(* Logix 5000 project; controller Drives_Line1 1756-L72 rev 20.13; software revision 20.04; part 13 of 21 *)
(* tags used below, declared in another part *)
   Bridle_01 : UDT_Bridle_3M;
   Entry_Accu : UDT_Entry_Accu;
   EntryConfig : UDT_Config_Zone;
   EntryCtrl : UDT_Control_Zone;
   EntrySetpoints : UDT_Setpoints_Zone;
   EntryStat : UDT_Status_Zone;
   In_Commands : UDT_Commands;
   In_Config : UDT_Config;
   In_Setpoints : UDT_Setpoints;
   LineCmd : UDT_Commands_Line;
   LineCtrl : UDT_Control_Line;
   LineStat : UDT_Status_Line;
   TM1 : UDT_TM;
   zConfigFromMaster : BOOL;

PROGRAM P16_Entry_Accu   (* main routine R00_Main *)
VAR
   ABS_01 : FBD_MATH_ADVANCED := (Source := -0.00068994303, Dest := 0.00068994303);
   BAND_01 : FBD_BOOLEAN_AND := (In3 := 1, In4 := 1, In5 := 1, In6 := 1, In7 := 1, In8 := 1);
   BAND_03 : FBD_BOOLEAN_AND := (In3 := 1, In4 := 1, In5 := 1, In6 := 1, In7 := 1, In8 := 1);
   BNOT_01 : FBD_BOOLEAN_NOT := (Out := 1);
   BNOT_02 : FBD_BOOLEAN_NOT := (In := 1);
   BNOT_04 : FBD_BOOLEAN_NOT := (Out := 1);
   BNOT_06 : FBD_BOOLEAN_NOT := (Out := 1);
   BOR_01 : FBD_BOOLEAN_OR;
   DIV_01 : FBD_MATH := (SourceA := -0.00068994303, SourceB := 4.0, Dest := -0.00017248576);
   DIV_02 : FBD_MATH;
   DIV_03 : FBD_MATH := (SourceA := 2.0441563, SourceB := 100.0, Dest := 0.020441564);
   DIV_04 : FBD_MATH := (SourceA := 0.5, SourceB := 4.0, Dest := 0.125);
   Entry_Accu_FBCounts_mm : DINT := 742;
   Entry_Accu_rev_mm : REAL := 0.1811;
   Exit_Accu_Rev_mm : REAL := 5.030181;
   IO_State_Exit_Accu : INT := 4;
   IO_State_Tmp_Exit_Accu : INT := 16384;
   MUL_01 : FBD_MATH := (SourceA := -2.9323564e-07, SourceB := 10865.999, Dest := -0.0031862983);
   MUL_02 : FBD_MATH := (SourceA := 2.0, SourceB := 2.0, Dest := 4.0);
   MUL_03 : FBD_MATH := (SourceA := 11670.0, SourceB := 742.0, Dest := 8659140.0);
   MUL_04 : FBD_MATH := (SourceB := 742.0);
   MUL_05 : FBD_MATH := (SourceA := 0.00034438504, SourceB := 0.5, Dest := 0.00017219252);
   MUL_06 : FBD_MATH := (SourceA := 1000.0, SourceB := 0.1811, Dest := 181.09999);
   MUL_07 : FBD_MATH := (SourceA := 181.09999, SourceB := 60.0, Dest := 10865.999);
   NEG_01 : FBD_MATH_ADVANCED := (Source := 50.0, Dest := -50.0);
   NEG_04 : FBD_MATH_ADVANCED := (Source := 0.02, Dest := -0.02);
   NEG_06 : FBD_MATH_ADVANCED := (Source := 0.020441564, Dest := -0.020441564);
   ons : BOOL[32];
   PI_01 : PROP_INT := (In := 23.319267, Initialize := 1, Kp := 25.0, Wld := 0.075, HighLimit := 100.0, ShapeKpPlus := 1.0, ShapeKpMinus := 1.0, ShapeWldPlus := 1.0, ShapeWldMinus := 1.0, RTSTime := 1, LowAlarm := 1, DeltaT := 0.05);
   PI_02 : PROP_INT := (In := -0.00033332407, Kp := 0.085, Wld := 0.01, HighLimit := 0.020441564, LowLimit := -0.020441564, ShapeKpPlus := 1.0, ShapeKpMinus := 1.0, ShapeWldPlus := 1.0, ShapeWldMinus := 1.0, RTSTime := 1, Out := 0.0003160029, DeltaT := 0.05);
   RLIM_01 : RATE_LIMITER := (In := -0.00017248576, IncRate := 0.5, DecRate := 0.5, RTSTime := 1, Out := -0.00017248576, DeltaT := 0.05);
   SCL_01 : SCALE := (In := 6033752.0, InRawMax := 8659140.0, InEUMax := 100.0, Out := 69.68073);
   SCL_02 : SCALE := (In := 6033752.0, InRawMax := 8659140.0, InEUMax := 11670.0, Out := 8131.741);
   SCL_03 : SCALE := (InRawMax := 100.0, Limiting := 1);
   SCL_04 : SCALE := (In := 5850.0, InRawMax := 30000.0, InEUMax := 1.0, Limiting := 1, Out := 0.19500001);
   SCL_05 : SCALE := (In := 5860.0, InRawMax := 30000.0, InEUMax := 1.0, Out := 0.19533333);
   SCL_08 : SCALE := (In := 0.00068994303, InRawMax := 0.125, InEUMax := 10.0, InEUMin := 2.0, Limiting := 1, Out := 2.0441563);
   SCRV_01 : S_CURVE := (Initialize := 1, AbsAlgRamp := 1, AccelRate := 0.04, DecelRate := 0.04, JerkRate := 0.25, RTSTime := 1, DeltaT := 0.05);
   SEL_01 : SELECT := (In1 := 50.0, In2 := 20.0, Out := 50.0);
   SSUM_01 : SELECTED_SUMMER := (In1 := 0.02, Gain1 := 1.0, In2 := -0.02, Gain2 := 1.0, Gain3 := 1.0, Select3 := 1, Gain4 := 1.0, Gain5 := 1.0, Gain6 := 1.0, Gain7 := 1.0, Gain8 := 1.0);
   SSUM_03 : SELECTED_SUMMER := (In1 := -0.00017248576, Gain1 := 1.0, Select1 := 1, Gain2 := 1.0, Gain3 := 1.0, Gain4 := 1.0, Gain5 := 1.0, Gain6 := 1.0, Gain7 := 1.0, Gain8 := 1.0, Out := -0.00017248576);
   SSUM_05 : SELECTED_SUMMER := (In1 := 0.00017219252, Gain1 := 1.0, Select1 := 1, In2 := -0.00017248576, Gain2 := 1.0, Select2 := 1, Gain3 := 1.0, Gain4 := 1.0, Gain5 := 1.0, Gain6 := 1.0, Gain7 := 1.0, Gain8 := 1.0, Out := -2.9323564e-07);
   SUB_01 : FBD_MATH := (SourceA := 93.0, SourceB := 69.68073, Dest := 23.319267);
   SUB_02 : FBD_MATH := (SourceA := 0.19500001, SourceB := 0.19533333, Dest := -0.00033332407);
   SUB_03 : FBD_MATH := (SourceB := 0.00068994303, Dest := -0.00068994303);
   SUB_04 : FBD_MATH := (SourceB := 0.00068994303, Dest := -0.00068994303);
   TofReset : TIMER := (PRE := 1000, ACC := 1000);
   TofTensionOnSp : TIMER := (PRE := 2500, ACC := 2500);
   TonNoResponse : TIMER := (PRE := 2500);
   TonRefOn : TIMER := (PRE := 750);
   TonTensionOnSp : TIMER := (PRE := 500, ACC := 549, EN := 1, DN := 1);
   zEntry_Accu_EncCounts : DINT := 4096;
   zEntry_Accu_Kp_Treg : REAL := 0.085;
   zEntry_Accu_MaxAccDec : REAL := 0.5;
   zEntry_Accu_Pos_PreLim : REAL := 100.0;
   zEntry_Accu_SpdRegMax : REAL := 50.0;
   zEntry_Accu_SpdRegMin : REAL := 20.0;
   zEntry_Accu_SpdTrim_HL : REAL := 10.0;
   zEntry_Accu_SpdTrim_LL : REAL := 2.0;
   zEntry_Accu_WLD_Treg : REAL := 0.01;
   zExit_Accu_Kp_Preg : REAL := 25.0;
   zExit_Accu_WLD_Preg : REAL := 0.075;
   zNoMaster : BOOL := 1;
   zTM1_Tens_Offset : REAL := 500.0;
END_VAR

ROUTINE R00_Main   (* ladder *)
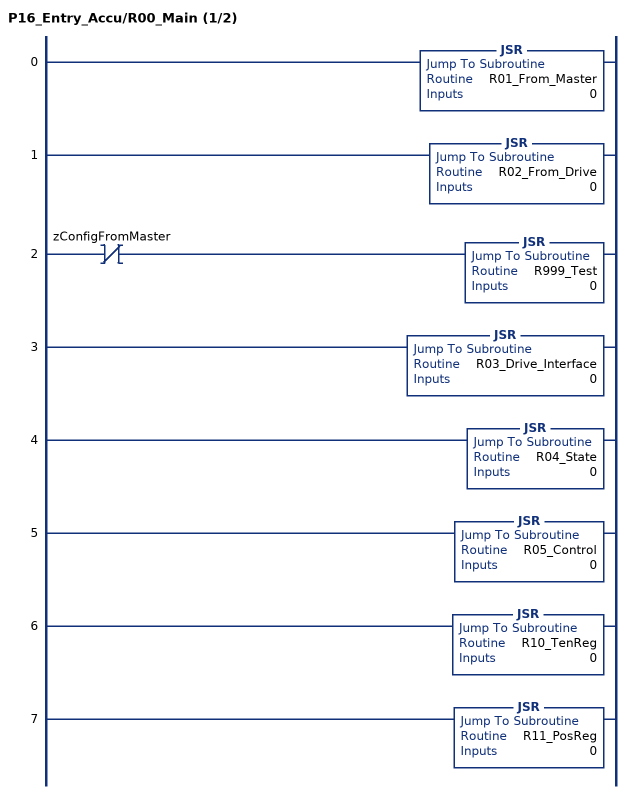
   0: JSR(R01_From_Master,0);
   1: JSR(R02_From_Drive,0);
   2: XIO(zConfigFromMaster)JSR(R999_Test,0);
   3: JSR(R03_Drive_Interface,0);
   4: JSR(R04_State,0);
   5: JSR(R05_Control,0);
   6: JSR(R10_TenReg,0);
   7: JSR(R11_PosReg,0);
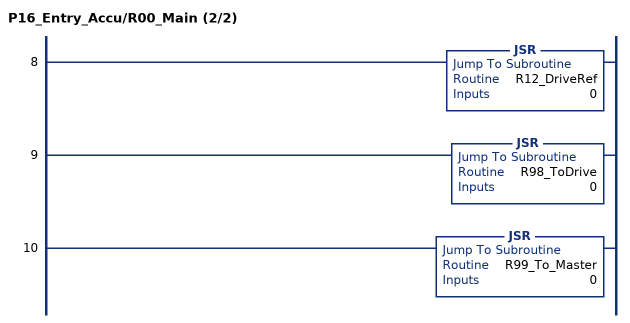
   8: JSR(R12_DriveRef,0);
   9: JSR(R98_ToDrive,0);
   10: JSR(R99_To_Master,0);
END_ROUTINE

ROUTINE R01_From_Master   (* ladder *)
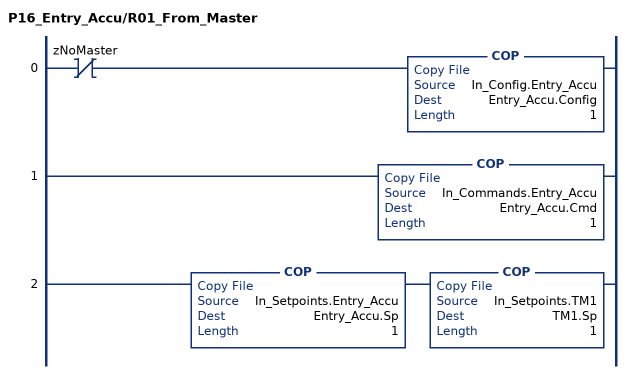
   0: XIO(zNoMaster)COP(In_Config.Entry_Accu,Entry_Accu.Config,1);
   1: COP(In_Commands.Entry_Accu,Entry_Accu.Cmd,1);
   2: COP(In_Setpoints.Entry_Accu,Entry_Accu.Sp,1)COP(In_Setpoints.TM1,TM1.Sp,1);
END_ROUTINE

ROUTINE R02_From_Drive   (* ladder *)
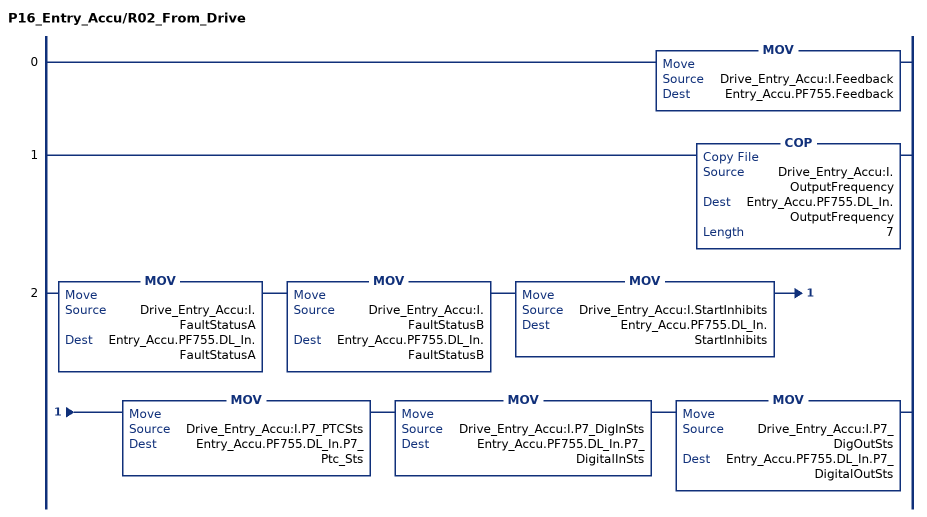
   0: MOV(Drive_Entry_Accu:I.Feedback,Entry_Accu.PF755.Feedback);
   1: COP(Drive_Entry_Accu:I.OutputFrequency,Entry_Accu.PF755.DL_In.OutputFrequency,7);
   2: MOV(Drive_Entry_Accu:I.FaultStatusA,Entry_Accu.PF755.DL_In.FaultStatusA)MOV(Drive_Entry_Accu:I.FaultStatusB,Entry_Accu.PF755.DL_In.FaultStatusB)MOV(Drive_Entry_Accu:I.StartInhibits,Entry_Accu.PF755.DL_In.StartInhibits)MOV(Drive_Entry_Accu:I.P7_PTCSts,Entry_Accu.PF755.DL_In.P7_Ptc_Sts)MOV(Drive_Entry_Accu:I.P7_DigInSts,Entry_Accu.PF755.DL_In.P7_DigitalInSts)MOV(Drive_Entry_Accu:I.P7_DigOutSts,Entry_Accu.PF755.DL_In.P7_DigitalOutSts);
END_ROUTINE

ROUTINE R03_Drive_Interface   (* ladder *)
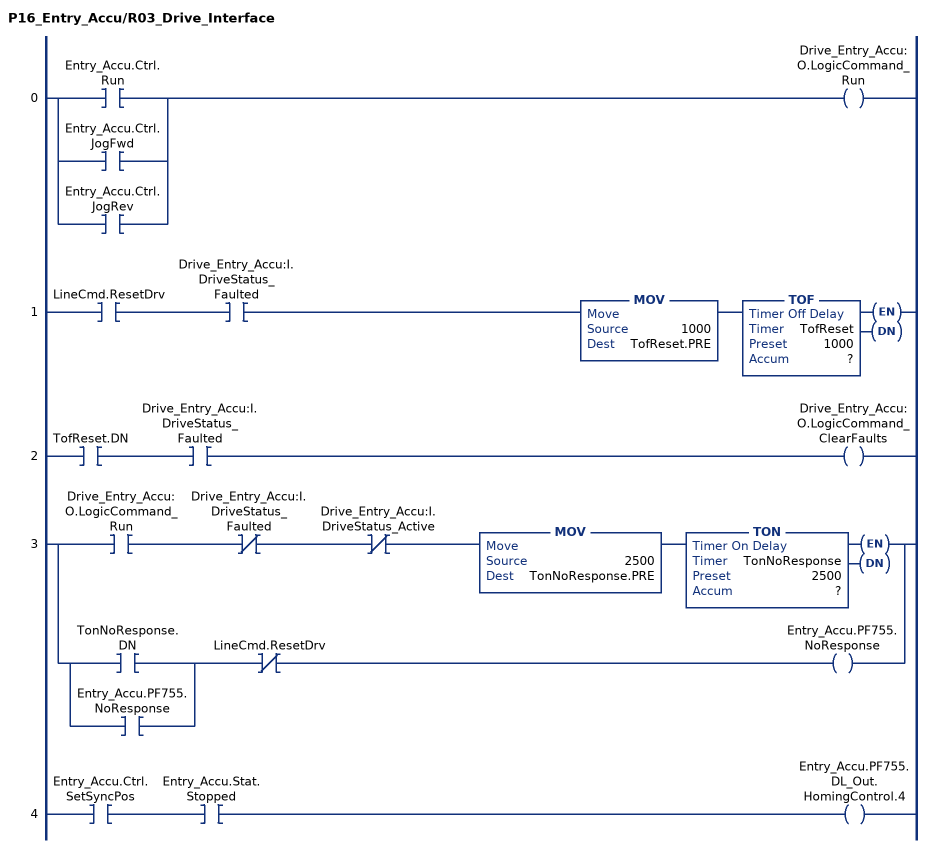
   0: [XIC(Entry_Accu.Ctrl.Run) ,XIC(Entry_Accu.Ctrl.JogFwd) ,XIC(Entry_Accu.Ctrl.JogRev) ]OTE(Drive_Entry_Accu:O.LogicCommand_Run);
   1: XIC(LineCmd.ResetDrv)XIC(Drive_Entry_Accu:I.DriveStatus_Faulted)MOV(1000,TofReset.PRE)TOF(TofReset,?,?);
   2: XIC(TofReset.DN)XIC(Drive_Entry_Accu:I.DriveStatus_Faulted)OTE(Drive_Entry_Accu:O.LogicCommand_ClearFaults);
   3: [XIC(Drive_Entry_Accu:O.LogicCommand_Run) XIO(Drive_Entry_Accu:I.DriveStatus_Faulted) XIO(Drive_Entry_Accu:I.DriveStatus_Active) MOV(2500,TonNoResponse.PRE) TON(TonNoResponse,?,?) ,[XIC(TonNoResponse.DN) ,XIC(Entry_Accu.PF755.NoResponse) ] XIO(LineCmd.ResetDrv) OTE(Entry_Accu.PF755.NoResponse) ];
   4: XIC(Entry_Accu.Ctrl.SetSyncPos)XIC(Entry_Accu.Stat.Stopped)OTE(Entry_Accu.PF755.DL_Out.HomingControl.4);
END_ROUTINE

ROUTINE R04_State   (* ladder *)
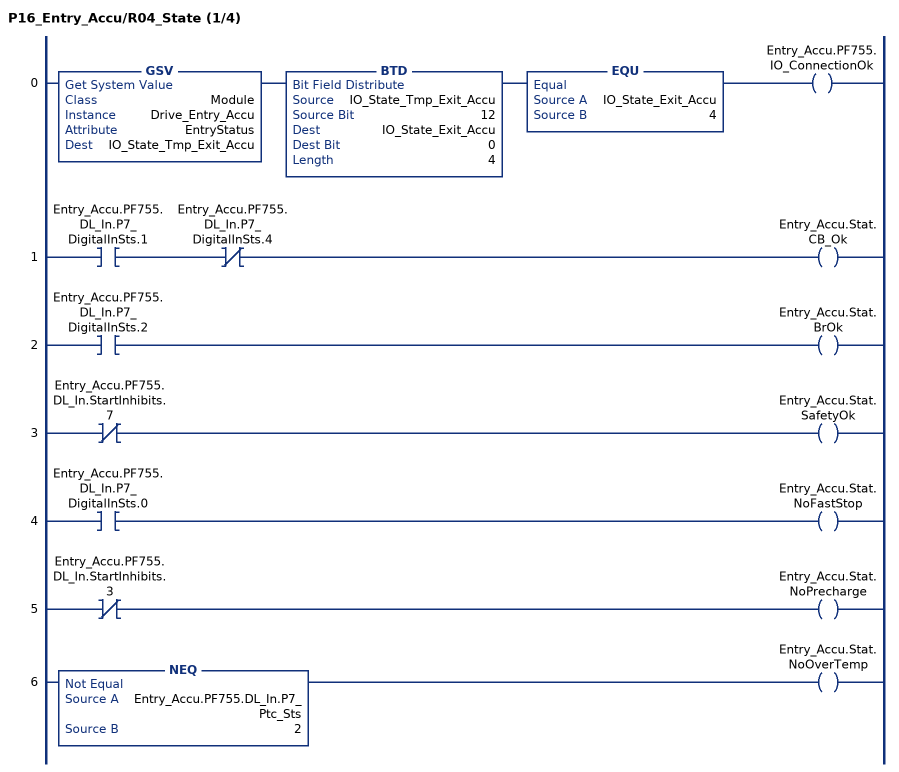
   0: GSV(Module,Drive_Entry_Accu,EntryStatus,IO_State_Tmp_Exit_Accu)BTD(IO_State_Tmp_Exit_Accu,12,IO_State_Exit_Accu,0,4)EQU(IO_State_Exit_Accu,4)OTE(Entry_Accu.PF755.IO_ConnectionOk);
   1: XIC(Entry_Accu.PF755.DL_In.P7_DigitalInSts.1)XIO(Entry_Accu.PF755.DL_In.P7_DigitalInSts.4)OTE(Entry_Accu.Stat.CB_Ok);
   2: XIC(Entry_Accu.PF755.DL_In.P7_DigitalInSts.2)OTE(Entry_Accu.Stat.BrOk);
   3: XIO(Entry_Accu.PF755.DL_In.StartInhibits.7)OTE(Entry_Accu.Stat.SafetyOk);
   4: XIC(Entry_Accu.PF755.DL_In.P7_DigitalInSts.0)OTE(Entry_Accu.Stat.NoFastStop);
   5: XIO(Entry_Accu.PF755.DL_In.StartInhibits.3)OTE(Entry_Accu.Stat.NoPrecharge);
   6: NEQ(Entry_Accu.PF755.DL_In.P7_Ptc_Sts,2)OTE(Entry_Accu.Stat.NoOverTemp);
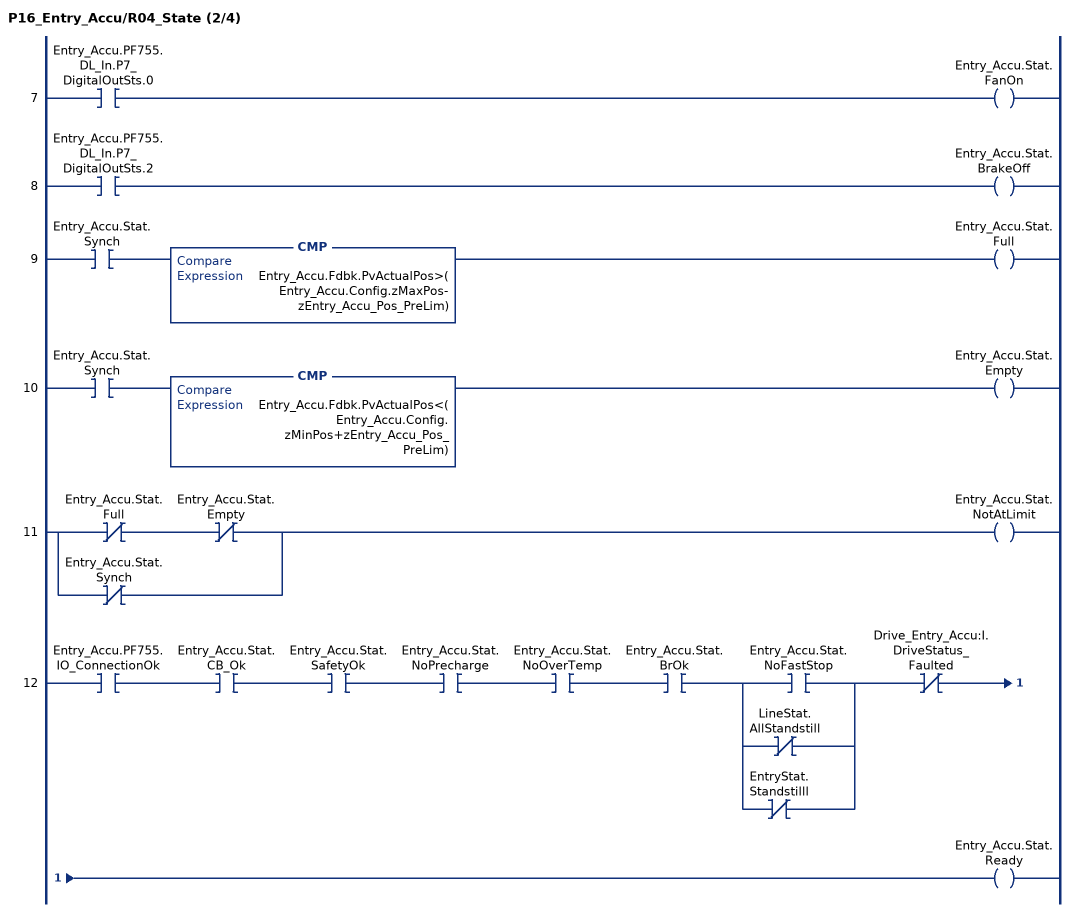
   7: XIC(Entry_Accu.PF755.DL_In.P7_DigitalOutSts.0)OTE(Entry_Accu.Stat.FanOn);
   8: XIC(Entry_Accu.PF755.DL_In.P7_DigitalOutSts.2)OTE(Entry_Accu.Stat.BrakeOff);
   9: XIC(Entry_Accu.Stat.Synch)CMP(Entry_Accu.Fdbk.PvActualPos>(Entry_Accu.Config.zMaxPos-zEntry_Accu_Pos_PreLim))OTE(Entry_Accu.Stat.Full);
   10: XIC(Entry_Accu.Stat.Synch)CMP(Entry_Accu.Fdbk.PvActualPos<(Entry_Accu.Config.zMinPos+zEntry_Accu_Pos_PreLim))OTE(Entry_Accu.Stat.Empty);
   11: [XIO(Entry_Accu.Stat.Full) XIO(Entry_Accu.Stat.Empty) ,XIO(Entry_Accu.Stat.Synch) ]OTE(Entry_Accu.Stat.NotAtLimit);
   12: XIC(Entry_Accu.PF755.IO_ConnectionOk)XIC(Entry_Accu.Stat.CB_Ok)XIC(Entry_Accu.Stat.SafetyOk)XIC(Entry_Accu.Stat.NoPrecharge)XIC(Entry_Accu.Stat.NoOverTemp)XIC(Entry_Accu.Stat.BrOk)[XIC(Entry_Accu.Stat.NoFastStop) ,XIO(LineStat.AllStandstill) ,XIO(EntryStat.Standstilll) ]XIO(Drive_Entry_Accu:I.DriveStatus_Faulted)OTE(Entry_Accu.Stat.Ready);
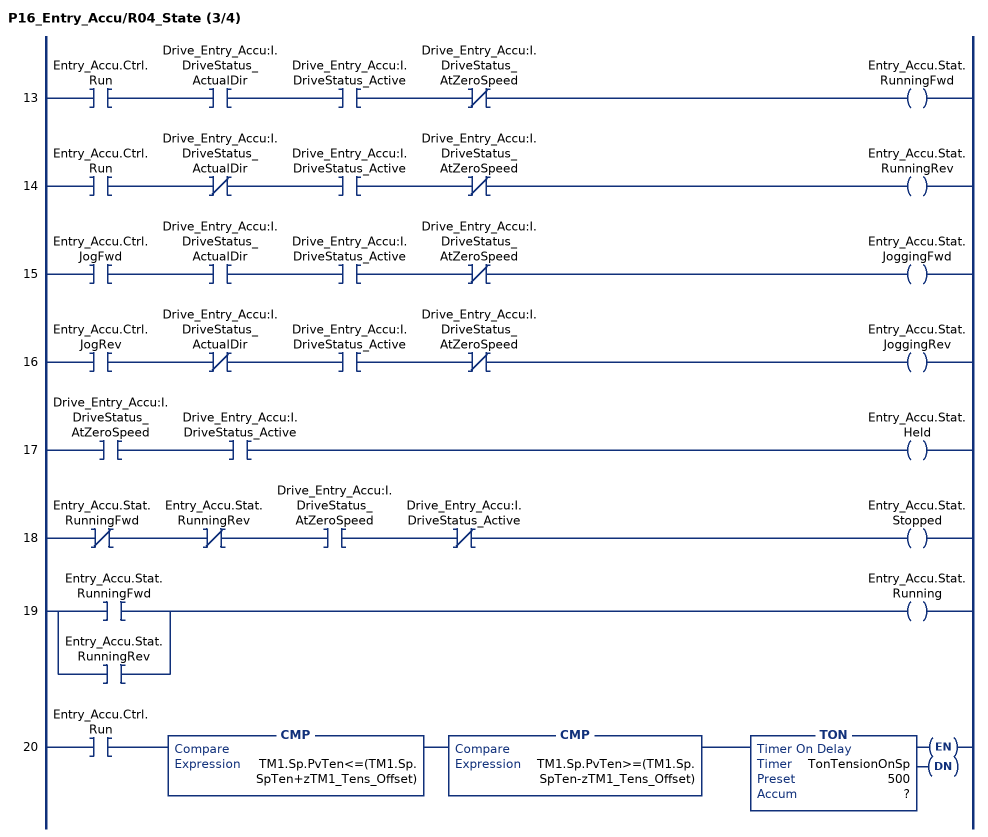
   13: XIC(Entry_Accu.Ctrl.Run)XIC(Drive_Entry_Accu:I.DriveStatus_ActualDir)XIC(Drive_Entry_Accu:I.DriveStatus_Active)XIO(Drive_Entry_Accu:I.DriveStatus_AtZeroSpeed)OTE(Entry_Accu.Stat.RunningFwd);
   14: XIC(Entry_Accu.Ctrl.Run)XIO(Drive_Entry_Accu:I.DriveStatus_ActualDir)XIC(Drive_Entry_Accu:I.DriveStatus_Active)XIO(Drive_Entry_Accu:I.DriveStatus_AtZeroSpeed)OTE(Entry_Accu.Stat.RunningRev);
   15: XIC(Entry_Accu.Ctrl.JogFwd)XIC(Drive_Entry_Accu:I.DriveStatus_ActualDir)XIC(Drive_Entry_Accu:I.DriveStatus_Active)XIO(Drive_Entry_Accu:I.DriveStatus_AtZeroSpeed)OTE(Entry_Accu.Stat.JoggingFwd);
   16: XIC(Entry_Accu.Ctrl.JogRev)XIO(Drive_Entry_Accu:I.DriveStatus_ActualDir)XIC(Drive_Entry_Accu:I.DriveStatus_Active)XIO(Drive_Entry_Accu:I.DriveStatus_AtZeroSpeed)OTE(Entry_Accu.Stat.JoggingRev);
   17: XIC(Drive_Entry_Accu:I.DriveStatus_AtZeroSpeed)XIC(Drive_Entry_Accu:I.DriveStatus_Active)OTE(Entry_Accu.Stat.Held);
   18: XIO(Entry_Accu.Stat.RunningFwd)XIO(Entry_Accu.Stat.RunningRev)XIC(Drive_Entry_Accu:I.DriveStatus_AtZeroSpeed)XIO(Drive_Entry_Accu:I.DriveStatus_Active)OTE(Entry_Accu.Stat.Stopped);
   19: [XIC(Entry_Accu.Stat.RunningFwd) ,XIC(Entry_Accu.Stat.RunningRev) ]OTE(Entry_Accu.Stat.Running);
   20: XIC(Entry_Accu.Ctrl.Run)CMP(TM1.Sp.PvTen<=(TM1.Sp.SpTen+zTM1_Tens_Offset))CMP(TM1.Sp.PvTen>=(TM1.Sp.SpTen-zTM1_Tens_Offset))TON(TonTensionOnSp,?,?);
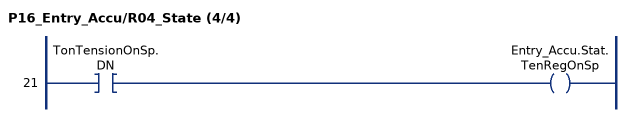
   21: XIC(TonTensionOnSp.DN)OTE(Entry_Accu.Stat.TenRegOnSp);
END_ROUTINE

ROUTINE R05_Control   (* ladder *)
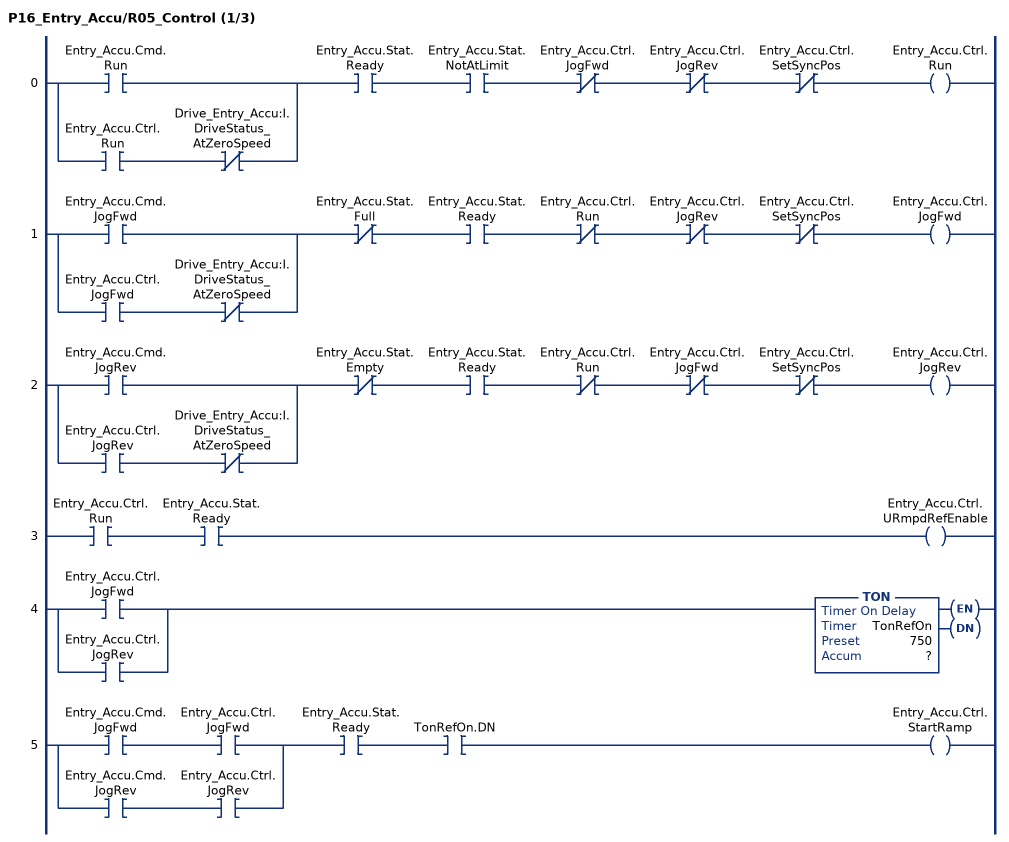
   0: [XIC(Entry_Accu.Cmd.Run) ,XIC(Entry_Accu.Ctrl.Run) XIO(Drive_Entry_Accu:I.DriveStatus_AtZeroSpeed) ]XIC(Entry_Accu.Stat.Ready)XIC(Entry_Accu.Stat.NotAtLimit)XIO(Entry_Accu.Ctrl.JogFwd)XIO(Entry_Accu.Ctrl.JogRev)XIO(Entry_Accu.Ctrl.SetSyncPos)OTE(Entry_Accu.Ctrl.Run);
   1: [XIC(Entry_Accu.Cmd.JogFwd) ,XIC(Entry_Accu.Ctrl.JogFwd) XIO(Drive_Entry_Accu:I.DriveStatus_AtZeroSpeed) ]XIO(Entry_Accu.Stat.Full)XIC(Entry_Accu.Stat.Ready)XIO(Entry_Accu.Ctrl.Run)XIO(Entry_Accu.Ctrl.JogRev)XIO(Entry_Accu.Ctrl.SetSyncPos)OTE(Entry_Accu.Ctrl.JogFwd);
   2: [XIC(Entry_Accu.Cmd.JogRev) ,XIC(Entry_Accu.Ctrl.JogRev) XIO(Drive_Entry_Accu:I.DriveStatus_AtZeroSpeed) ]XIO(Entry_Accu.Stat.Empty)XIC(Entry_Accu.Stat.Ready)XIO(Entry_Accu.Ctrl.Run)XIO(Entry_Accu.Ctrl.JogFwd)XIO(Entry_Accu.Ctrl.SetSyncPos)OTE(Entry_Accu.Ctrl.JogRev);
   3: XIC(Entry_Accu.Ctrl.Run)XIC(Entry_Accu.Stat.Ready)OTE(Entry_Accu.Ctrl.URmpdRefEnable);
   4: [XIC(Entry_Accu.Ctrl.JogFwd) ,XIC(Entry_Accu.Ctrl.JogRev) ]TON(TonRefOn,?,?);
   5: [XIC(Entry_Accu.Cmd.JogFwd) XIC(Entry_Accu.Ctrl.JogFwd) ,XIC(Entry_Accu.Cmd.JogRev) XIC(Entry_Accu.Ctrl.JogRev) ]XIC(Entry_Accu.Stat.Ready)XIC(TonRefOn.DN)OTE(Entry_Accu.Ctrl.StartRamp);
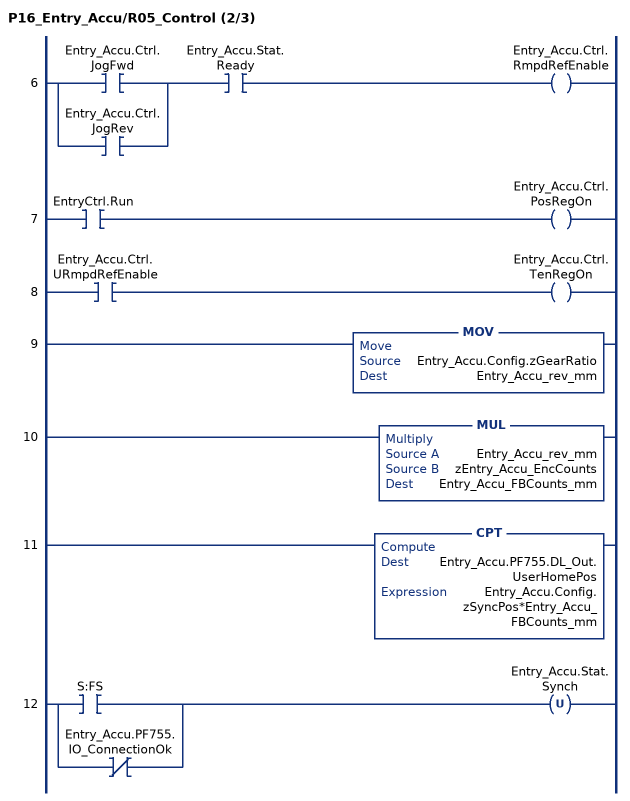
   6: [XIC(Entry_Accu.Ctrl.JogFwd) ,XIC(Entry_Accu.Ctrl.JogRev) ]XIC(Entry_Accu.Stat.Ready)OTE(Entry_Accu.Ctrl.RmpdRefEnable);
   7: XIC(EntryCtrl.Run)OTE(Entry_Accu.Ctrl.PosRegOn);
   8: XIC(Entry_Accu.Ctrl.URmpdRefEnable)OTE(Entry_Accu.Ctrl.TenRegOn);
   9: MOV(Entry_Accu.Config.zGearRatio,Entry_Accu_rev_mm);
   10: MUL(Entry_Accu_rev_mm,zEntry_Accu_EncCounts,Entry_Accu_FBCounts_mm);
   11: CPT(Entry_Accu.PF755.DL_Out.UserHomePos,Entry_Accu.Config.zSyncPos*Entry_Accu_FBCounts_mm);
   12: [XIC(S:FS) ,XIO(Entry_Accu.PF755.IO_ConnectionOk) ]OTU(Entry_Accu.Stat.Synch);
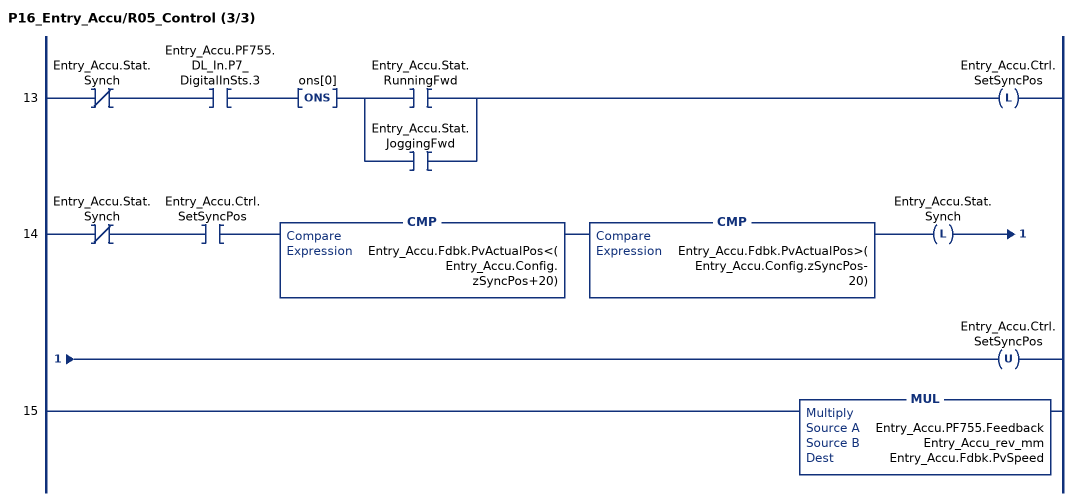
   13: XIO(Entry_Accu.Stat.Synch)XIC(Entry_Accu.PF755.DL_In.P7_DigitalInSts.3)ONS(ons[0])[XIC(Entry_Accu.Stat.RunningFwd) ,XIC(Entry_Accu.Stat.JoggingFwd) ]OTL(Entry_Accu.Ctrl.SetSyncPos);
   14: XIO(Entry_Accu.Stat.Synch)XIC(Entry_Accu.Ctrl.SetSyncPos)CMP(Entry_Accu.Fdbk.PvActualPos<(Entry_Accu.Config.zSyncPos+20))CMP(Entry_Accu.Fdbk.PvActualPos>(Entry_Accu.Config.zSyncPos-20))OTL(Entry_Accu.Stat.Synch)OTU(Entry_Accu.Ctrl.SetSyncPos);
   15: MUL(Entry_Accu.PF755.Feedback,Entry_Accu_rev_mm,Entry_Accu.Fdbk.PvSpeed);
END_ROUTINE

ROUTINE R10_TenReg   (* function block diagram *)
   SHEET 1   // Scale setpoint
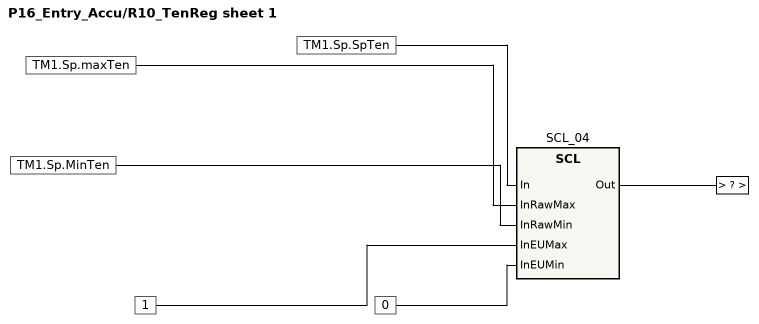
   SCL_04 : SCL(In := TM1.Sp.SpTen, InRawMax := TM1.Sp.maxTen, InRawMin := TM1.Sp.MinTen, InEUMax := 1, InEUMin := 0);
   WIRE(?) := SCL_04.Out;
   SHEET 2   // Scale tension feedback
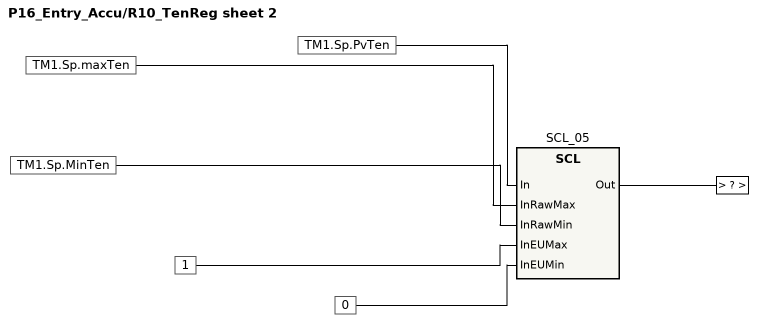
   SCL_05 : SCL(In := TM1.Sp.PvTen, InRawMax := TM1.Sp.maxTen, InRawMin := TM1.Sp.MinTen, InEUMax := 1, InEUMin := 0);
   WIRE(?) := SCL_05.Out;
   SHEET 3   // Trim limits
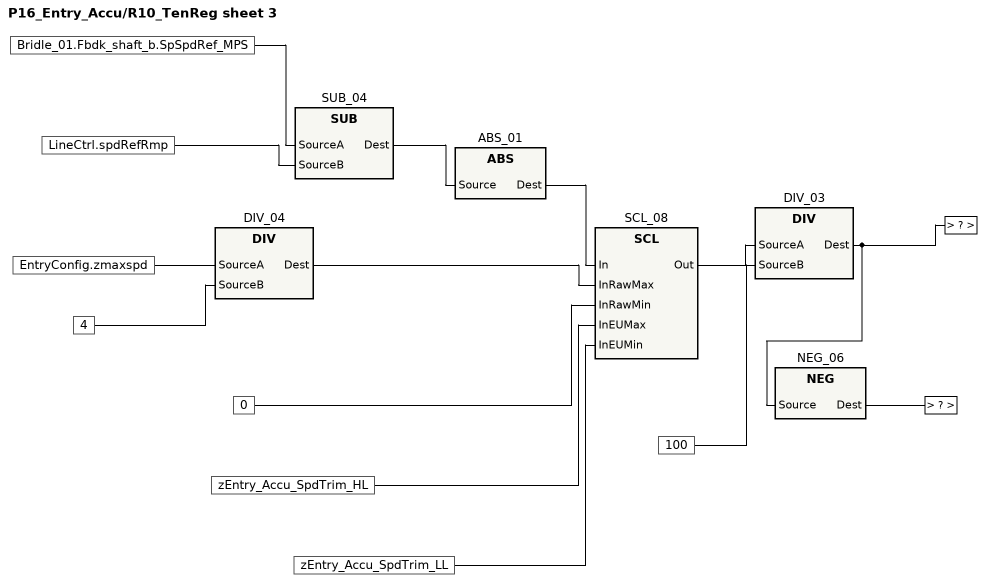
   DIV_04 : DIV(SourceA := EntryConfig.zmaxspd, SourceB := 4);
   SUB_04 : SUB(SourceA := Bridle_01.Fbdk_shaft_b.SpSpdRef_MPS, SourceB := LineCtrl.spdRefRmp);
   ABS_01 : ABS(Source := SUB_04.Dest);
   SCL_08 : SCL(In := ABS_01.Dest, InRawMax := DIV_04.Dest, InRawMin := 0, InEUMax := zEntry_Accu_SpdTrim_HL, InEUMin := zEntry_Accu_SpdTrim_LL);
   DIV_03 : DIV(SourceA := SCL_08.Out, SourceB := 100);
   NEG_06 : NEG(Source := DIV_03.Dest);
   WIRE(?) := NEG_06.Dest;
   WIRE(?) := DIV_03.Dest;
   SHEET 4   // Tension regulator
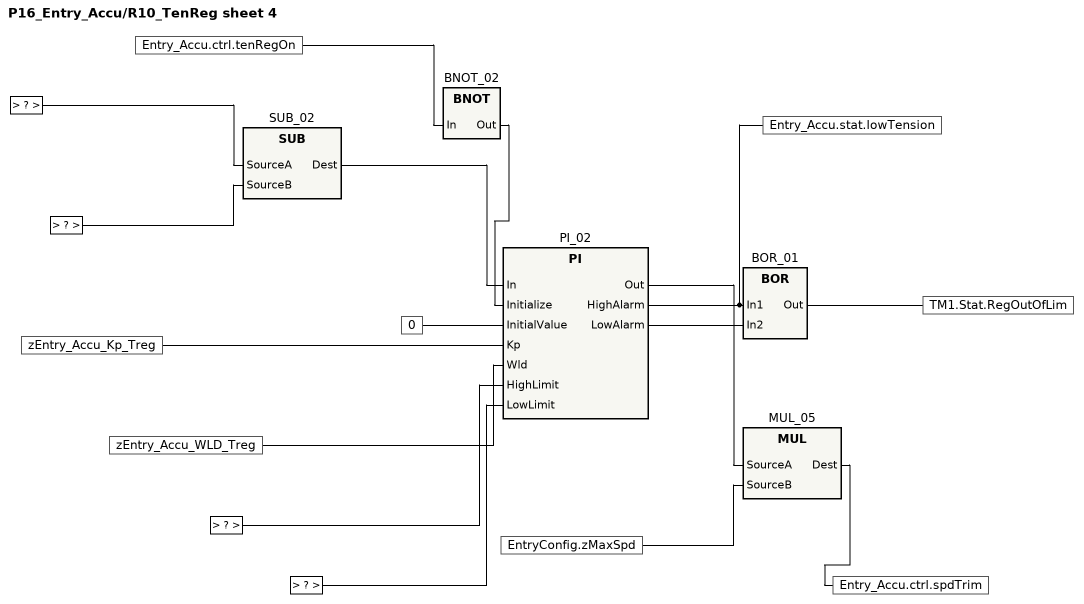
   SUB_02 : SUB(SourceA := WIRE(?), SourceB := WIRE(?));
   BNOT_02 : BNOT(In := Entry_Accu.ctrl.tenRegOn);
   PI_02 : PI(In := SUB_02.Dest, Initialize := BNOT_02.Out, InitialValue := 0, Kp := zEntry_Accu_Kp_Treg, Wld := zEntry_Accu_WLD_Treg, HighLimit := WIRE(?), LowLimit := WIRE(?));
   BOR_01 : BOR(In1 := PI_02.HighAlarm, In2 := PI_02.LowAlarm);
   MUL_05 : MUL(SourceA := PI_02.Out, SourceB := EntryConfig.zMaxSpd);
   Entry_Accu.stat.lowTension := PI_02.HighAlarm;
   Entry_Accu.ctrl.spdTrim := MUL_05.Dest;
   TM1.Stat.RegOutOfLim := BOR_01.Out;
END_ROUTINE

ROUTINE R11_PosReg   (* function block diagram *)
   SHEET 1   // Scale feedback
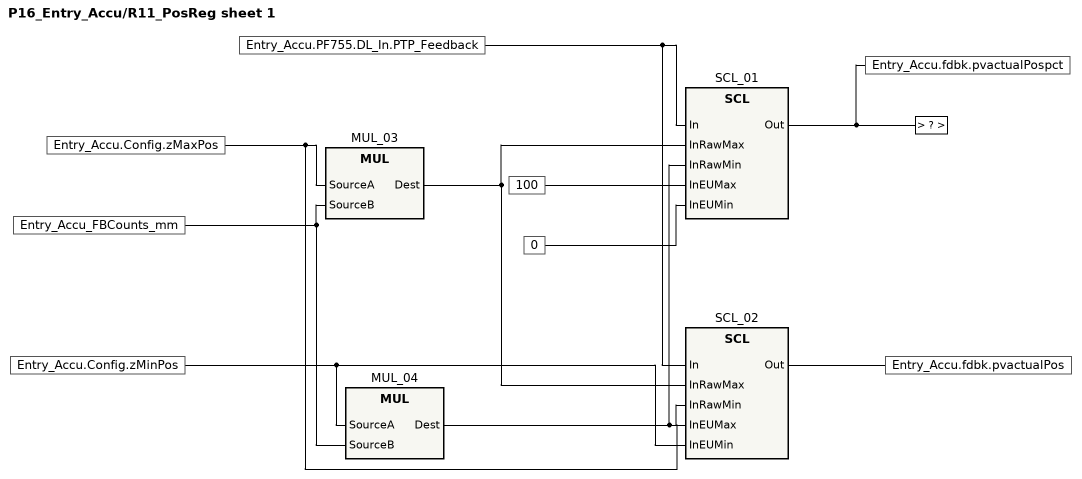
   MUL_03 : MUL(SourceA := Entry_Accu.Config.zMaxPos, SourceB := Entry_Accu_FBCounts_mm);
   MUL_04 : MUL(SourceA := Entry_Accu.Config.zMinPos, SourceB := Entry_Accu_FBCounts_mm);
   SCL_01 : SCL(In := Entry_Accu.PF755.DL_In.PTP_Feedback, InRawMax := MUL_03.Dest, InRawMin := MUL_04.Dest, InEUMax := 100, InEUMin := 0);
   SCL_02 : SCL(In := Entry_Accu.PF755.DL_In.PTP_Feedback, InRawMax := MUL_03.Dest, InRawMin := MUL_04.Dest, InEUMax := Entry_Accu.Config.zMaxPos, InEUMin := Entry_Accu.Config.zMinPos);
   Entry_Accu.fdbk.pvactualPospct := SCL_01.Out;
   Entry_Accu.fdbk.pvactualPos := SCL_02.Out;
   WIRE(?) := SCL_01.Out;
   SHEET 2   // Position regulator
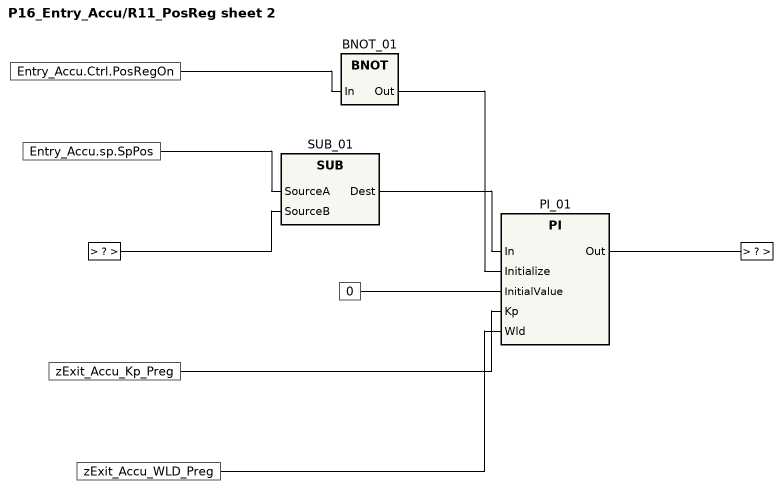
   BNOT_01 : BNOT(In := Entry_Accu.Ctrl.PosRegOn);
   SUB_01 : SUB(SourceA := Entry_Accu.sp.SpPos, SourceB := WIRE(?));
   PI_01 : PI(In := SUB_01.Dest, Initialize := BNOT_01.Out, InitialValue := 0, Kp := zExit_Accu_Kp_Preg, Wld := zExit_Accu_WLD_Preg);
   WIRE(?) := PI_01.Out;
   SHEET 3   // Scale position regulator output
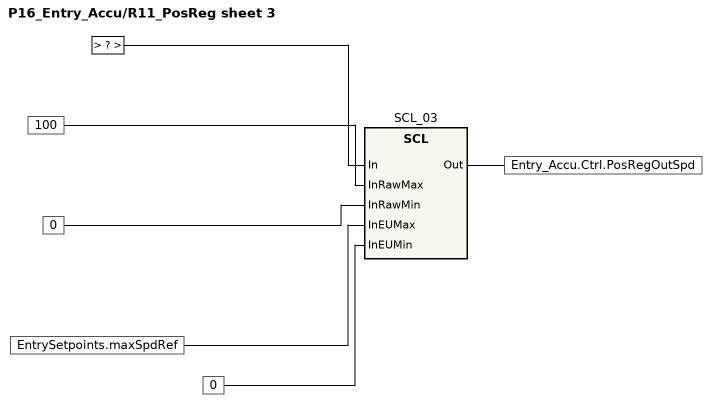
   SCL_03 : SCL(In := WIRE(?), InRawMax := 100, InRawMin := 0, InEUMax := EntrySetpoints.maxSpdRef, InEUMin := 0);
   Entry_Accu.Ctrl.PosRegOutSpd := SCL_03.Out;
END_ROUTINE
